(*
Nazwa:			E_LidSealingState
Opis:			Stan wbijania nasadek
Wersja:			v0.1
Data:			2018-10-10
Autor:			TW
Urzadzenia:		
Konfiguracja:	
Info:
*)

TYPE E_CapPushingState :
(               	
	eReady:=1,				//Gotowość
	ePushing:=2,			//Wbijanie
	eHolding:=3,			//Przytrzymywanie
	ePushed:=4,				//Wbito
	eGoingUp:=5			//Podnoszenie
);
END_TYPE

(* stored: Version 1.1.0.1, ProductVersion 3.1.4026.13, FileIdentifier 1a63c2fbded6d53221b3c96c58df9882ad55fdfe, FileSignature 8655c769c6a8cffcd58405cc31ed5fc2e0bcc12187ea41cc788a8b1ae41bb3d41f315536f23552ed4abe3af57b154f575fa675c60faa53301a28703a02e5230228f0a4f4d660b66f422441a4ce1aa7c7f27a19802d960118cba96bb1baecee7a57ab12c4d83a8b33927f8658ea7421c008eb238ca7f9860e7a1cca48a384d857b736419efd78efebdb83e764f1ca3bb1665923630179fc384171233d00eacc3be7cb0e4163ff1b95474e846979940355ea6faaf002d24bac97fe0741b59607d86f106cffcab3426f1ecf4190eaa5864182d0ae8c86cc213a79a279fdc2b01484a2f9ab4a4747dddfb96879e2d710f8014155fe43e3342215614ef32a7aefc65e
   DUT E_CapPushingState: Id {fbbfeea5-63c8-4dd9-aff0-7153796f801a} *)
